PROGRAM P_Demo_F_BA_IsLeapYear
VAR
    argNYear                       : UDINT                          := 0; // nYear
    fnReturn                       : BOOL; // 返回值
END_VAR

// =============================================================================
// Tc3_BA2_Common.F_BA_IsLeapYear 演示程序
// =============================================================================
// 场景：日历显示控件按年份生成"2 月有几天"。
//
// 价值：一行 FC 替代手写 `(y MOD 4 = 0 AND y MOD 100 <> 0) OR (y MOD 400 = 0)` —— 易写错。
//
// 验证：登录 PLC 后，按例程内变量在线写值；监视输出 / 返回值，结合 §1 功能
//       简述的预期行为对照（详见配套 .md 文档 §7 业务场景）。
//
// 验证步骤：
//   1. 右键 PLC 项目下 POUs 文件夹 → Add → Existing Item → 选本 .TcPOU 文件
//   2. 引用 Tc3_BA2_Common（References → Add library）
//   3. 编译 → 登录 → 运行；按上方『验证』指引在线写值观察
// =============================================================================

fnReturn := F_BA_IsLeapYear(
    nYear                    := argNYear
);

END_PROGRAM

(* stored: Version 1.1.0.1, ProductVersion 3.1.4024.5
   POU P_Demo_F_BA_IsLeapYear: Id {1985fa1e-ee97-5b69-8998-30c35979f309}, SpecialFunc None *)
